// TwinCAT 3 PLC project PLC1
// ProgramVersion: 3.1.4024.0
// libraries:
//   Tc2_MC2, * (Beckhoff Automation GmbH)
//   Tc2_Standard, * (Beckhoff Automation GmbH)
//   Tc2_System, * (Beckhoff Automation GmbH)
//   Tc3_Module, * (Beckhoff Automation GmbH)
// project tree:
//   GVLs/ GVL.TcGVL
//   / PlcTask.TcTTO
//   POUs/ Halt_Axis.TcPOU, Jog_Axis.TcPOU, MAIN.TcPOU, Move_Axis_Absolute.TcPOU, Move_Axis_Velocity.TcPOU
// real-time tasks:
//   TASK PlcTask: cycle T#10ms, priority 20, ADS port 350
// motion (NC):
//   TASK NC-Task 1 SAF: cycle T#2ms, priority 4, ADS port 501
//   TASK NC-Task 1 SVB: cycle T#10ms, priority 8, ADS port 511
//   AXIS Asse Virtuale (id 1)
//     OtherSettings: AllowMotionCmdToSlave=true
//     encoder EncType=1
//     drive DrvType=5
//       Analog: TorqueSetpointScale=10, ScaleFactorActTorque=0.1
//       TimeComp: TaskDelayCycles=1
//     controller CtrType=1
//       CtrPara: PriorControlFactor=1
//         Observer: BandWidth=20
// variable links:
//   PLC1/PLC1 Instance <-> NC-Task 1 SAF/Axes/Asse Virtuale
//     PlcTask Inputs/GVL.Axis.NcToPlc <-> Outputs/ToPlc
//     PlcTask Outputs/GVL.Axis.PlcToNc <-> Inputs/FromPlc

CONFIGURATION PLC1
    RESOURCE PLC ON TwinCAT3
        TASK PlcTask(INTERVAL := T#10ms, PRIORITY := 20);
        PROGRAM MAIN WITH PlcTask : MAIN;
    END_RESOURCE
END_CONFIGURATION

// ---- GVLs/GVL.TcGVL
{attribute 'qualified_only'}
VAR_GLOBAL
	Axis: AXIS_REF;
END_VAR

// ---- POUs/MAIN.TcPOU
PROGRAM MAIN
VAR
	fbPower: MC_Power;
	AxisEnabled: BOOL;
	EnableAxis: BOOL;
	fbReadStatus: MC_ReadStatus;
END_VAR

EnableAxisAction();
ReadAxisStatus();
Jog_Axis();
Halt_Axis();
Move_Axis_Velocity();
Move_Axis_Absolute();

ACTION EnableAxisAction:
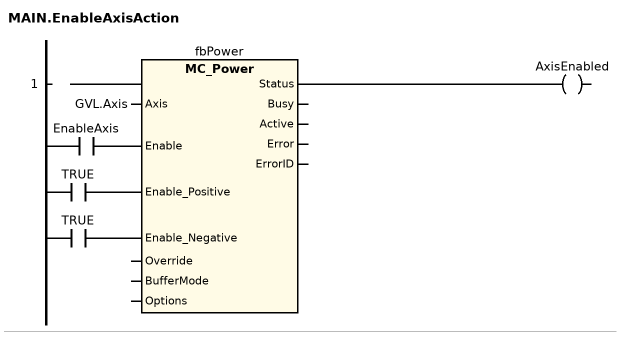
// NETWORK 1
fbPower(Axis := GVL.Axis, Enable := EnableAxis, Enable_Positive := TRUE, Enable_Negative := TRUE); // MC_Power
AxisEnabled := fbPower.Status;
END_ACTION

ACTION ReadAxisStatus:
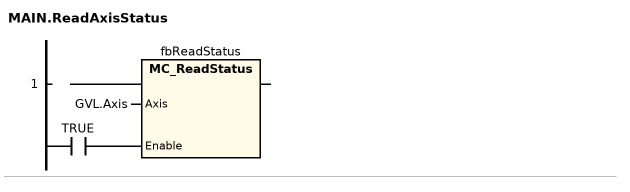
// NETWORK 1
fbReadStatus(Axis := GVL.Axis, Enable := TRUE); // MC_ReadStatus
END_ACTION

END_PROGRAM

// ---- POUs/Jog_Axis.TcPOU
PROGRAM Jog_Axis
VAR
	fbJog: MC_Jog;
	JogForwardPB: BOOL;
	JogBackwardsPB: BOOL;
END_VAR

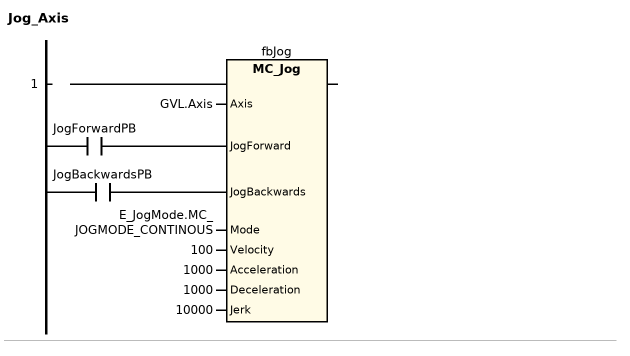
// NETWORK 1
fbJog(
    Axis := GVL.Axis,
    JogForward := JogForwardPB,
    JogBackwards := JogBackwardsPB,
    Mode := E_JogMode.MC_JOGMODE_CONTINOUS,
    Velocity := 100,
    Acceleration := 1000,
    Deceleration := 1000,
    Jerk := 10000); // MC_Jog

END_PROGRAM

// ---- POUs/Halt_Axis.TcPOU
PROGRAM Halt_Axis
VAR
	fbHalt: MC_Halt;
	HaltPB: BOOL;
	HaltDone: BOOL;
END_VAR

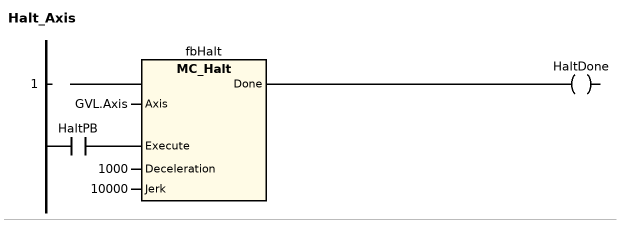
// NETWORK 1
fbHalt(Axis := GVL.Axis, Execute := HaltPB, Deceleration := 1000, Jerk := 10000); // MC_Halt
HaltDone := fbHalt.Done;

END_PROGRAM

// ---- POUs/Move_Axis_Velocity.TcPOU
PROGRAM Move_Axis_Velocity
VAR
	fbMoveVelocity: MC_MoveVelocity;
	MoveVelocityExecute: BOOL;
	InVelocity: BOOL;
END_VAR

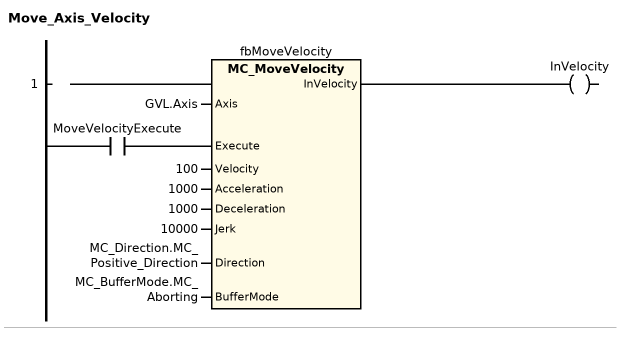
// NETWORK 1
fbMoveVelocity(
    Axis := GVL.Axis,
    Execute := MoveVelocityExecute,
    Velocity := 100,
    Acceleration := 1000,
    Deceleration := 1000,
    Jerk := 10000,
    Direction := MC_Direction.MC_Positive_Direction,
    BufferMode := MC_BufferMode.MC_Aborting); // MC_MoveVelocity
InVelocity := fbMoveVelocity.InVelocity;

END_PROGRAM

// ---- POUs/Move_Axis_Absolute.TcPOU
PROGRAM Move_Axis_Absolute
VAR
	fbMoveAbsolute: MC_MoveAbsolute;
	MoveAbsoluteExecute: BOOL;
	Position: LREAL := 1000;
	Done: BOOL;
END_VAR

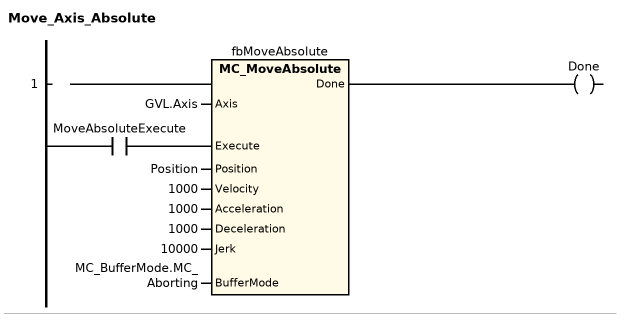
// NETWORK 1
fbMoveAbsolute(
    Axis := GVL.Axis,
    Execute := MoveAbsoluteExecute,
    Position := Position,
    Velocity := 1000,
    Acceleration := 1000,
    Deceleration := 1000,
    Jerk := 10000,
    BufferMode := MC_BufferMode.MC_Aborting); // MC_MoveAbsolute
Done := fbMoveAbsolute.Done;

END_PROGRAM
